# EPICS substitutions: iocs/omsIOC/iocBoot/iocOms/MAXv.substitutions
file "$(MOTOR)/db/motor.db"
{
pattern
{P,     N,  M,        DTYP,        C,  S,  DESC,           EGU,  DIR,  VELO,  VBAS,  ACCL,  BDST,  BVEL,  BACC,  MRES,    PREC,  DHLM,  DLLM,  INIT}
{oms:,  1,  "m$(N)",  "OMS MAXv",  0,  0,  "MAXv M$(N)",   mm,   Pos,  1,     .1,    .2,    0,     1,     .2,    2.5e-4,  5,     100,   -100,  ""}
{oms:,  2,  "m$(N)",  "OMS MAXv",  0,  1,  "MAXv M$(N)",   mm,   Pos,  1,     .1,    .2,    0,     1,     .2,    2.5e-4,  5,     100,   -100,  ""}
{oms:,  3,  "m$(N)",  "OMS MAXv",  0,  2,  "MAXv M$(N)",   mm,   Pos,  1,     .1,    .2,    0,     1,     .2,    2.5e-4,  5,     100,   -100,  ""}
{oms:,  4,  "m$(N)",  "OMS MAXv",  0,  3,  "MAXv M$(N)",   mm,   Pos,  1,     .1,    .2,    0,     1,     .2,    2.5e-4,  5,     100,   -100,  ""}
{oms:,  5,  "m$(N)",  "OMS MAXv",  0,  4,  "MAXv M$(N)",   mm,   Pos,  1,     .1,    .2,    0,     1,     .2,    2.5e-4,  5,     100,   -100,  ""}
{oms:,  6,  "m$(N)",  "OMS MAXv",  0,  5,  "MAXv M$(N)",   mm,   Pos,  1,     .1,    .2,    0,     1,     .2,    2.5e-4,  5,     100,   -100,  ""}
{oms:,  7,  "m$(N)",  "OMS MAXv",  0,  6,  "MAXv M$(N)",   mm,   Pos,  1,     .1,    .2,    0,     1,     .2,    2.5e-4,  5,     100,   -100,  ""}
{oms:,  8,  "m$(N)",  "OMS MAXv",  0,  7,  "MAXv M$(N)",   mm,   Pos,  1,     .1,    .2,    0,     1,     .2,    2.5e-4,  5,     100,   -100,  ""}
}
